PROGRAM P_InfluxDataCollector
VAR 
	Data : REFERENCE TO ST_DATA := P_UpdateDAQ.DataDaq;  
	Tick : LREAL; 
	ActualBufferTime : TIME; 
	
	InfluxData : FB_InfluxDataCollector; 

	Timer1Hz 	: TON; 
	Timer10Hz 	: TON; 
	Timer100Hz 	: TON; 	

END_VAR

Tick := Tick + 1;
RunTimers(); 

// ========= Initialize Data
	InfluxData.Initialize( 	HostName 		:= 'MachinePLC',			// <<---- 	Change to Descriptive MachinePLC name, eg: MachinePLC_TLU 
							Database 		:= 'RD',			// <<---- 	Change to Database name. Needs to be setup beforehand.
							Measurement 	:= 'CKD_Test');	// <<---- 	Measurentname in database. Eg: LORCHALT
// ========= Add Data tags.
// These are written to each "point" i.e. for each ms.
// Add eg: Current State of TestBench - for easy search later on
															
	//Data.AddTag('State','Default');						

// ========= Add Actual Data

	InfluxData.AddLreal('Tick', Tick);

// ======== 1 Hz Data
	IF Time_1Hz THEN
		InfluxData.AddLreal('Test1Hz', 1);	
	
		InfluxAddData_1Hz(		Data 			:= Data,
								DataCollector 	:=  InfluxData); 	
						
	END_IF
	
// ======== 10 Hz Data
	IF Time_10Hz THEN
		InfluxData.AddLreal('Test10Hz', 10);
	
		InfluxAddData_10Hz(	Data 			:= Data,
								DataCollector 	:=  InfluxData); 		
		
	END_IF

// ======== 100 Hz Data
	IF Time_100Hz THEN
		InfluxData.AddLreal('Test100Hz', 100);
	
		InfluxAddData_100Hz(	Data 			:= Data,
								DataCollector 	:=  InfluxData); 

		InfluxAddData_1000Hz(	Data 			:= Data,
								DataCollector 	:=  InfluxData); 
	
								
	END_IF


// =========== Add TimeStamp and start new "point"
InfluxData.AddTimeStamp(ActualBufferTime => ActualBufferTime); 















ResetTimersIfDone();

METHOD ResetTimersIfDone : BOOL
IF Timer1Hz.Q THEN
	Timer1Hz(IN := FALSE); 
	Timer1Hz(IN := TRUE); 

END_IF
IF Timer10Hz.Q THEN
	Timer10Hz(IN := FALSE); 
	Timer10Hz(IN := TRUE); 
	

END_IF
IF Timer100Hz.Q THEN
	Timer100Hz(IN := FALSE); 
	Timer100Hz(IN := TRUE); 
	
END_IF
END_METHOD

METHOD RunTimers : BOOL
Timer1Hz(	IN := TRUE, PT := T#1S		); 
Timer10Hz(	IN := TRUE, PT := T#100MS	); 
Timer100Hz(	IN := TRUE, PT := T#10MS	);
END_METHOD

PROPERTY Time_100Hz : BOOL
GET
Time_100Hz := Timer100Hz.Q;
END_GET
END_PROPERTY

PROPERTY Time_10Hz : BOOL
GET
Time_10Hz := Timer10Hz.Q;
END_GET
END_PROPERTY

PROPERTY Time_1Hz : BOOL
GET
Time_1Hz := Timer1Hz.Q;
END_GET
END_PROPERTY

END_PROGRAM

(* stored: Version 1.1.0.1, ProductVersion 3.1.4022.11
   POU P_InfluxDataCollector: Id {5890daa8-c4a5-4cdf-a905-3dfb235d7713}, SpecialFunc None
   Method ResetTimersIfDone: Id {961ce8e5-b526-4f59-bf7a-6a7c37564e66}
   Method RunTimers: Id {6e2b8f82-2805-4145-9c6b-f3dcfa4c82bb}
   Property Time_100Hz: Id {a94ea9fd-eea9-40d1-bc5f-e9174e0989ab}
   Get Get: Id {7871c46d-dc5c-4542-9256-e2a59dd9f15b}
   Property Time_10Hz: Id {9fdde1d8-45d3-4afc-85b5-fbefe968ea8b}
   Get Get: Id {fecd4283-c36b-4303-a2dd-2adb5c157d15}
   Property Time_1Hz: Id {d11ea6bf-5130-4225-b2bb-274eeedeb585}
   Get Get: Id {0685c72b-5e74-4d07-bff6-eb6598f00475} *)
